FUNCTION_BLOCK BoolValuesTest EXTENDS TcUnit.FB_TestSuite
VAR
END_VAR

FalseBoolValue();
TrueBoolValue();

METHOD FalseBoolValue : BOOL
VAR
	value : FalseBoolValue;
END_VAR
TcUnit.TEST('Get false bool value');

AssertEquals_BOOL(
	Expected := FALSE,
	Actual := value.Value,
	Message := 'FalseBoolValue should return FALSE value');

TEST_FINISHED();
END_METHOD

METHOD TrueBoolValue : BOOL
VAR
	value : TrueBoolValue;
END_VAR
TcUnit.TEST('Get true bool value');

AssertEquals_BOOL(
	Expected := TRUE,
	Actual := value.Value,
	Message := 'TrueBoolValue should return TRUE value');

TEST_FINISHED();
END_METHOD

END_FUNCTION_BLOCK

(* stored: Version 1.1.0.1, ProductVersion 3.1.4024.15
   POU BoolValuesTest: Id {47c75fac-3a1d-091a-21c9-fa02f37d83cd}, SpecialFunc None
   Method FalseBoolValue: Id {1f3a4816-c10a-0590-30cb-e56e765cdb99}
   Method TrueBoolValue: Id {b81252c0-63f8-03fe-3fac-d80941b090ab} *)
